TYPE typePoints :
STRUCT
	PointXTime:ULINT;
	PointYValue:REAL;
END_STRUCT
END_TYPE

(* stored: Version 1.1.0.1, ProductVersion 3.1.4024.11
   DUT typePoints: Id {ee777055-b216-0b4a-1d96-4da1876aef66} *)
